// TIA Portal project "Sim1" (V15)

(* hardware
DEVICE "S7-1200 station_1"  S7-1200 Station
   slot 0: "Rack_0"  S7-1200 Rack  Rack  V1.0
   slot 1: "PLC_1"  CPU 1214C DC/DC/DC  6ES7 214-1AG40-0XB0  V4.2
   slot 3: "AQ 1x12BIT_1"  AQ1 signal board  6ES7 232-4HA30-0XB0  V1.0
   slot 101: "CM 1243-5"  CM 1243-5  6GK7 243-5DX30-0XE0  V1.3
   slot 102: "CM 1241 (RS485)_1"  CM 1241 (RS485)  6ES7 241-1CH30-0XB0  V1.0
*)

// ===== PLC "PLC_1"  CPU 1214C DC/DC/DC =====

VAR_GLOBAL   // PLC tag table "Default tag table"
   ""start1"" AT %I0.0 : Bool;
   ""start2"" AT %I0.1 : Bool;
   ""start3"" AT %I0.4 : Bool;
   ""start5"" AT %I0.5 : Bool;
   ""wyjscie1"" AT %Q0.0 : Bool;
   ""WY_1"" AT %Q0.2 : Bool;
   ""WY"" AT %Q0.3 : Bool;
   ""wyjscie5"" AT %Q0.5 : Bool;
END_VAR